FUNCTION_BLOCK EventSelect (* Basic Function Block Type *)
  (* Standard: 61499-2 *)
  (* Version 0.2, 2003-12-04, JHC, Rockwell Automation, Renamed for better indexing. *)
  (* Version 0.1, 2002-11-05, JHC, Rockwell Automation, Corrected missing ST element in Algorithm REQ. *)
  (* Version 0.0, 2000-05-30, JHC, Rockwell Automation *)
  (* Compiler header: package fb.rt.template; *)
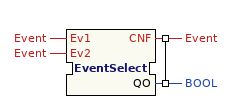
  EVENT_INPUT
    Ev1; (* Normal Execution Request *)
    Ev2;
  END_EVENT
  EVENT_OUTPUT
    CNF WITH QO; (* Execution Confirmation *)
  END_EVENT
  VAR_OUTPUT
    QO : BOOL; (* Output event qualifier *)
  END_VAR
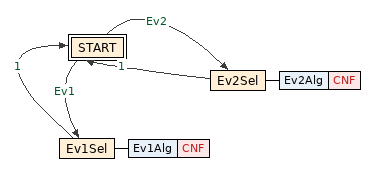
  EC_STATES
    START; (* Initial State *)
    Ev1Sel : Ev1Alg -> CNF; (* Normal execution *)
    Ev2Sel : Ev2Alg -> CNF;
  END_STATES
  EC_TRANSITIONS
    START TO Ev1Sel := Ev1;
    Ev1Sel TO START := 1;
    START TO Ev2Sel := Ev2;
    Ev2Sel TO START := 1;
  END_TRANSITIONS
  ALGORITHM INIT IN ST: (* Initialization algorithm *)

  END_ALGORITHM
  ALGORITHM Ev1Alg IN ST: (* Normally executed algorithm *)
QO:=TRUE;
  END_ALGORITHM
  ALGORITHM Ev2Alg IN ST:
QO:=FALSE;
  END_ALGORITHM
END_FUNCTION_BLOCK
